{attribute 'reflection'}
FUNCTION_BLOCK Mediator
VAR_INPUT

	MoverArray				: ARRAY [1..Param.MAX_MOVERS] OF POINTER TO Mover;
	
	MoverListArray			: ARRAY [0..Param.MAX_MOVERLISTS-1] OF POINTER TO MoverList;
	PositionTriggerArray	: ARRAY [0..Param.MAX_POSITIONTRIGGERS-1] OF POINTER TO PositionTrigger;
	StationArray			: ARRAY [0..Param.MAX_STATIONS-1] OF POINTER TO Station;
	ZoneArray				: ARRAY [0..Param.MAX_ZONES-1] OF POINTER TO Zone;
	TrackArray				: ARRAY [0..Param.NUM_TRACKS] OF POINTER TO Track;	// track 0 is a special absolute case, this makes the array 1 larger than normal	

	GROUP_REF				: AXES_GROUP_REF;
	
END_VAR
VAR_OUTPUT
	Error			: BOOL;			// error is currently active
	ErrorID			: UDINT;		// errorID of the active error
	ErrorOrigin		: STRING;		// error source, in case of errored internal function block
	NumMovers		: USINT;		// number of movers in system
END_VAR
VAR
	{attribute 'instance-path'}
	{attribute 'noinit'}
	{attribute 'hide'}
	internalInstancePath		: STRING;	// instance naming, for diagnostics purposes

	internalMoverList				: MoverList;
	internalMoverListRecalc			: BOOL;
	internalM1DetectFlag			: BOOL;
	internalM1DetectState			: INT;
	internalEnableGroupFlag			: BOOL;
	internalEnableGroupState		: INT;
	internalEnabled					: BOOL;
	internalMover1Error				: BOOL;
	
	// implements memoization of Mediator.AllMotorModulesReady
	// so it is only computed once per scan when needed
	internalMotorModuleEnabled		:  MotorModuleStatus_typ;
	internalMotorModule48v			:  MotorModuleStatus_typ;

	// ========= XTS Utility Diagnostics =========
	fbXtsEnvironment				: FB_TcIoXtsEnvironment;
	fbXtsEnvironmentVisu			: FB_XtsEnvironmentVisu;
	nEnvironmentState				: INT;
	internalInfoServerOTCID			: UDINT;

	internalEnvironment				: I_TcIoXtsEnvironment;
	internalXPU						: I_TcIoXtsProcessingUnit;
	internalInfoServer				: I_TcIoXtsInfoServer;
	internalInfoServerCount			: UINT;
	
	// ========= internal function blocks =========
	fbGroupStatus			: MC_GroupReadStatus;
	fbGroupEnable			: MC_GroupEnable;
	fbGroupReset			: MC_GroupReset;
	fbGroupStop				: MC_GroupStop;

END_VAR
VAR CONSTANT
	ADD_TO_GROUP_SIZE		: UDINT := 30;
END_VAR

METHOD AddMover : BOOL
VAR_INPUT
	
	Mover		: REFERENCE TO Mover;

END_VAR

VAR
	duplicateFound		: BOOL;
	i					: DINT;
	emptyIDX			: DINT := -1;;
END_VAR


// Check for duplicates

IF __ISVALIDREF( Mover ) THEN
	
	Mover.Mediator			REF= THIS^;

	duplicateFound			:= FALSE;
	
	FOR i := 1 TO SIZEOF( MoverArray ) / SIZEOF( MoverArray[1] ) DO
		IF MoverArray[i] <> 0 THEN		// verify the element is clear to prevent overwrites
			IF ADR(Mover) = MoverArray[i] THEN
				duplicateFound		:= TRUE;	// this mover is already mediated
			END_IF
		ELSE
			// track the first empty index
			IF (emptyIDX = -1) THEN
				emptyIDX	:= i;
			END_IF;
		END_IF	
	END_FOR
	
	// if no empty index is available set a message and return
	IF emptyIDX = -1 THEN
		ADSLOGSTR( ADSLOG_MSGTYPE_WARN, 'AddMover System Array is full. %s not added. Check Params.MAX_MOVERS' , Mover.InstancePath);
		RETURN;
	END_IF;
	
	IF duplicateFound = FALSE THEN
		
		THIS^.MoverArray[emptyIDX]		:= ADR( Mover );	// new mover into empty array element

		// Automatically register the mover with any Position Triggers
		FOR i := 0 TO SIZEOF( PositionTriggerArray ) / SIZEOF( PositionTriggerArray[0] ) - 1 DO
			IF PositionTriggerArray[i] <> 0 THEN
				PositionTriggerArray[i]^.RegisterMover( Mover );
			END_IF			
		END_FOR
		
		// Automatically register the mover with any Zones
		FOR i := 0 TO SIZEOF( ZoneArray ) / SIZEOF( ZoneArray[0] ) - 1 DO
			IF ZoneArray[i] <> 0 THEN
				ZoneArray[i]^.RegisterMover( Mover );
			END_IF
		END_FOR
		
	END_IF
END_IF

// set the flag to recalculate the internal mover list
internalMoverListRecalc := TRUE;
END_METHOD

METHOD AddMoverList : BOOL
VAR_INPUT
	
	MoverList		: REFERENCE TO MoverList;

END_VAR

VAR
	duplicateFound		: BOOL;
	i					: DINT;
	emptyIDX			: DINT := -1;
END_VAR


// Check for duplicates
IF __ISVALIDREF( MoverList ) THEN
	
	MoverList.Mediator			REF= THIS^;
	
	duplicateFound				:= FALSE;
	
	FOR i := 0 TO SIZEOF( MoverListArray ) / SIZEOF( MoverListArray[0] ) - 1 DO
		IF MoverListArray[i] <> 0 THEN		// verify the element is clear to prevent overwrites
			IF ADR( MoverList ) = MoverListArray[i] THEN
				duplicateFound		:= TRUE;		// this moverlist is already mediated
			END_IF
		ELSE
			// track the first empty index
			IF (emptyIDX = -1) THEN
				emptyIDX	:= i;
			END_IF;
		END_IF
	END_FOR
	
	// if no empty index is available set a message and return
	IF emptyIDX = -1 THEN
		ADSLOGSTR( ADSLOG_MSGTYPE_WARN, 'MoverList System Array is full. %s not added. Check Params.MAX_MOVERLISTS' , MoverList.InstancePath);
		RETURN;
	END_IF;
	
	IF duplicateFound = FALSE THEN
		THIS^.MoverListArray[emptyIDX]		:= ADR( MoverList );
	END_IF
END_IF

// set the flag to recalculate the internal mover list
internalMoverListRecalc := TRUE;
END_METHOD

METHOD AddPositionTrigger : BOOL
VAR_INPUT
	
	PositionTrigger		: REFERENCE TO PositionTrigger;

END_VAR

VAR
	duplicateFound		: BOOL;
	i					: DINT;
	emptyIDX			: DINT := -1;
END_VAR


// Check for duplicates
IF __ISVALIDREF( PositionTrigger ) THEN
	
	PositionTrigger.Mediator		REF= THIS^;
	
	duplicateFound					:= FALSE;
	
	FOR i := 0 TO SIZEOF( PositionTriggerArray ) / SIZEOF( PositionTriggerArray[0] ) - 1 DO
		IF PositionTriggerArray[i] <> 0 THEN		// verify the element is clear to prevent overwrites
			IF ADR( PositionTrigger ) = PositionTriggerArray[i] THEN
				duplicateFound		:= TRUE;		// this moverlist is already mediated
			END_IF
		ELSE
			// track the first empty index
			IF (emptyIDX = -1) THEN
				emptyIDX	:= i;
			END_IF;
		END_IF
	END_FOR
	
	// if no empty index is available set a message and return
	IF emptyIDX = -1 THEN
		ADSLOGSTR( ADSLOG_MSGTYPE_WARN, 'AddPositionTrigger System Array is full. %s not added. Check Params.MAX_POSITIONTRIGGERS' , PositionTrigger.InstancePath);
		RETURN;
	END_IF;
	
	IF duplicateFound = FALSE THEN
		THIS^.PositionTriggerArray[emptyIDX]		:= ADR( PositionTrigger );
		
		// Automatically register all existing movers with the new position trigger
		FOR i := 1 TO SIZEOF( MoverArray ) / SIZEOF( MoverArray[1] ) DO
			IF MoverArray[i] <> 0 THEN
				THIS^.PositionTriggerArray[emptyIDX]^.RegisterMover( MoverArray[i]^ );
			END_IF
		END_FOR		
		
	END_IF
END_IF
END_METHOD

METHOD AddStation : BOOL
VAR_INPUT
	
	Station		: REFERENCE TO Station;

END_VAR

VAR
	duplicateFound		: BOOL;
	i					: DINT;
	emptyIDX			: DINT := -1;
END_VAR


// Check for duplicates
IF __ISVALIDREF( Station ) THEN
	
	Station.Mediator	REF= THIS^;
	
	duplicateFound		:= FALSE;
	
	FOR i := 0 TO SIZEOF( StationArray ) / SIZEOF( StationArray[0] ) - 1 DO
		IF StationArray[i] <> 0 THEN		// verify the element is clear to prevent overwrites
			IF ADR( Station ) = StationArray[i] THEN
				duplicateFound		:= TRUE;		// this moverlist is already mediated
			END_IF
		ELSE
			// track the first empty index
			IF (emptyIDX = -1) THEN
				emptyIDX	:= i;
			END_IF;
		END_IF
	END_FOR
	
	// if no empty index is available set a message and return
	IF emptyIDX = -1 THEN
		ADSLOGSTR( ADSLOG_MSGTYPE_WARN, 'AddStation System Array is full. %s not added. Check Params.MAX_STATIONS' , Station.InstancePath);
		RETURN;
	END_IF;
	
	IF duplicateFound = FALSE THEN
		THIS^.StationArray[emptyIDX]		:= ADR( Station );
		// store unique index for station
		Station.Id := emptyIDX;
	END_IF
END_IF
END_METHOD

METHOD AddTrack : BOOL
VAR_INPUT
	
	Track		: REFERENCE TO Track;

END_VAR

VAR
	duplicateFound		: BOOL;
	i					: UDINT;
	emptyIDX			: UDINT;
END_VAR


// Check for duplicates
IF __ISVALIDREF( Track ) THEN
	
	Track.Mediator		REF= THIS^;
	
	duplicateFound		:= FALSE;
	
	FOR i := 0 TO SIZEOF( TrackArray ) / SIZEOF( TrackArray[0] ) - 1 DO
		IF TrackArray[i] <> 0 THEN		// verify the element is clear to prevent overwrites
			IF ADR( Track ) = TrackArray[i] THEN
				duplicateFound		:= TRUE;		// this moverlist is already mediated
			END_IF
		ELSE
			// track the first empty index
			IF (emptyIDX = 0) THEN
				emptyIDX	:= i;
			END_IF;
		END_IF
	END_FOR
	
	IF duplicateFound = FALSE THEN
		THIS^.TrackArray[emptyIDX]		:= ADR( Track );
	END_IF
END_IF
END_METHOD

METHOD AddZone : BOOL
VAR_INPUT
	
	Zone		: REFERENCE TO Zone;

END_VAR

VAR
	duplicateFound		: BOOL;
	i					: DINT;
	emptyIDX			: DINT := -1;
END_VAR


// Check for duplicates
IF __ISVALIDREF( Zone ) THEN
	
	Zone.Mediator		REF= THIS^;
	
	duplicateFound		:= FALSE;
	
	FOR i := 0 TO SIZEOF( ZoneArray ) / SIZEOF( ZoneArray[0] ) - 1 DO
		IF ZoneArray[i] <> 0 THEN		// verify the element is clear to prevent overwrites
			IF ADR( Zone ) = ZoneArray[i] THEN
				duplicateFound		:= TRUE;		// this moverlist is already mediated
			END_IF
		ELSE
			// track the first empty index
			IF (emptyIDX = -1) THEN
				emptyIDX	:= i;
			END_IF;
		END_IF
	END_FOR
	
	// if no empty index is available set a message and return
	IF emptyIDX = -1 THEN
		ADSLOGSTR( ADSLOG_MSGTYPE_WARN, 'AddZone System Array is full. %s not added. Check Params.MAX_ZONES' , Zone.InstancePath);
		RETURN;
	END_IF;
	
	IF duplicateFound = FALSE THEN
		THIS^.ZoneArray[emptyIDX]		:= ADR( Zone );
		
		// Automatically register all existing movers with the new zone
		FOR i := 1 TO SIZEOF( MoverArray ) / SIZEOF( MoverArray[1] ) DO
			IF MoverArray[i] <> 0 THEN
				THIS^.ZoneArray[emptyIDX]^.RegisterMover( MoverArray[i]^ );
			END_IF
		END_FOR
		
	END_IF
END_IF
END_METHOD

{attribute 'monitoring' := 'call'}
PROPERTY AllMotorModules48vReady : Bool
GET
VAR
	I				: UDINT;
	nParts			: UDINT;
	b48vReady	: BOOL;
	PartTcIo		: I_TcIoXtsXpuPart;
END_VAR
// this is calculation and ADS intensive so the result is memozied once per scan

// only run the sum if the calc bit has not been set for this scan
IF (NOT internalMotorModule48v.calcComplete) THEN
	// Monitor DriveStatus to disallow motion commands before high drive has been achieved.
	IF fbXtsEnvironment.P_IsInitialized THEN
	// Get number of parts. 
		nParts:= fbXtsEnvironment.XpuTcIo(1).P_PartCount;
		IF nParts <> 0 THEN
			// Get number of modules per part and check their state
			b48vReady:= TRUE;
			FOR I := 1 TO nParts DO 
				PartTcIo := fbXtsEnvironment.XpuTcIo(1).PartTcIo(UDINT_TO_UINT(I));
				// and the previous result with the result for this part
				b48vReady := b48vReady AND PartMotorModules48vReady(PartTcIo);
			END_FOR
		END_IF
	END_IF

	// memoize the result
	internalMotorModule48v.calcResult := b48vReady;
	internalMotorModule48v.calcComplete := TRUE;
END_IF;

// return the result
AllMotorModules48vReady:= internalMotorModule48v.calcResult;
END_GET
END_PROPERTY

{attribute 'monitoring' := 'call'}
PROPERTY AllMotorModulesEnabled : Bool
GET
VAR
	I				: UDINT;
	nParts			: UDINT;
	bHighDriveReady	: BOOL;
	PartTcIo		: I_TcIoXtsXpuPart;
END_VAR
// this is calculation and ADS intensive so the result is memozied once per scan

// only run the sum if the calc bit has not been set for this scan
IF (NOT internalMotorModuleEnabled.calcComplete) THEN
	// Monitor DriveStatus to disallow motion commands before high drive has been achieved.
	IF fbXtsEnvironment.P_IsInitialized THEN
	// Get number of parts. 
		nParts:= fbXtsEnvironment.XpuTcIo(1).P_PartCount;
		IF nParts <> 0 THEN
			// Get number of modules per part and check their state
			bHighDriveReady:= TRUE;
			FOR I := 1 TO nParts DO 
				PartTcIo := fbXtsEnvironment.XpuTcIo(1).PartTcIo(UDINT_TO_UINT(I));
				// and the previous result with the result for this part
				bHighDriveReady := bHighDriveReady AND PartMotorModulesEnabled(PartTcIo);
			END_FOR
		END_IF
	END_IF

	// memoize the result
	internalMotorModuleEnabled.calcResult := bHighDriveReady;
	internalMotorModuleEnabled.calcComplete := TRUE;
END_IF;

// return the result
AllMotorModulesEnabled:= internalMotorModuleEnabled.calcResult;
END_GET
END_PROPERTY

PROPERTY CompleteMoverList : iMoverList
GET
VAR
	i: UDINT;
END_VAR
// the mover list is populated in cyclic when needed
// flags in the methods .AddMover and .AddMoverList trigger the recalculation

CompleteMoverList	:= internalMoverList;
END_GET
END_PROPERTY

METHOD Cyclic : BOOL
VAR_INPUT
	NUM_MOVERS			: USINT;
END_VAR

VAR
	eMoverIdDetectionMode : MoverIdDetectionMode;
	eMoverIdDetectionState : MoverIdDetectionStateEnum;
END_VAR

VAR_INST
	MsgCreate		: FB_TcMessage;
	
	// station info state machine support
	nInfoServerState : INT;
	PartStartEnd : ARRAY [1..Param.PART_ARRAY_SIZE] OF ARRAY [0..1] OF LREAL;
	nPartsInTrack1	: UDINT;
	TrackPartInfo	: ARRAY[1..TcIoXtsEnvironmentParameterList.MaxPartsPerTrack] OF ST_PartInfoItems;
	PartInfo 		: St_PartInfoItems;
	nInfoServerStations		: UDINT;
	nUsableStations			: UDINT;
	StationTcIo		: I_TcIoXtsInfoServerInfoStation;
	nStationPartNum	: UDINT;
	pXtsStation		: POINTER TO Station;
	PartObjectIds	: ARRAY [1..TcIoXtsEnvironmentParameterList.MaxXtsPartsPerXpu] OF OTCID;
	StopPositions	: ARRAY [1..TcIoXtsEnvironmentParameterList.MaxXtsStopPositionsPerStation] OF LREAL := [0.0];
	i				: UDINT;
	j				: UDINT;
	workingStation	: UDINT;
	
	XPUDetectionState	: DetectionStateEnum;
END_VAR
// this method contains multiple state machines denoted by the headers below

// update output data
NumMovers := NUM_MOVERS;

// clear memoized values for recalculation
internalMotorModuleEnabled.calcComplete := FALSE;
internalMotorModule48v.calcComplete := FALSE;

// regenerate the internal mover list when necessary
IF (internalMoverListRecalc) THEN
	// this is returned by the property CompleteMoverList, and does not need to be calculated on every call to the property
	// reset flag
	internalMoverListRecalc := FALSE;
	// clear the list
	internalMoverList.UnregisterAll();
	// re-populate the list
	FOR i := 1 TO SIZEOF( MoverArray ) / SIZEOF( MoverArray[1] ) DO
		IF MoverArray[i] <> 0 THEN
			internalMoverList.RegisterMover( MoverArray[i]^ );
		END_IF
	END_FOR
END_IF

// Handle all project cyclic calls

FOR i := 1 TO Param.MAX_MOVERS DO
	IF MoverArray[i] <> 0 THEN
		// handle cyclic calls
		MoverArray[i]^.Cyclic( GROUP_REF );			// could make this ca group addition clener
		MoverArray[i]^.AxisReference.ReadStatus();
		MoverArray[i]^.MoverIndex := i;
	END_IF
END_FOR

FOR i := 0 TO Param.MAX_STATIONS - 1 DO
	IF StationArray[i] <> 0 THEN
		StationArray[i]^.Cyclic();
	END_IF
END_FOR

FOR i := 0 TO Param.MAX_POSITIONTRIGGERS - 1 DO
	IF PositionTriggerArray[i] <> 0 THEN
		PositionTriggerArray[i]^.Cyclic();
	END_IF
END_FOR

FOR i := 0 TO Param.NUM_TRACKS DO
	IF TrackArray[i] <> 0 THEN
		TrackArray[i]^.Cyclic();
	END_IF
END_FOR

// *************************************************************************
// environment state machine
// *************************************************************************

CASE nEnvironmentState OF
	0:	// ----------------------------------------- Enable Init Items
	
		// the procedure for initializing the XTS environment has changed
		// this step previously held configuration values for the environment
		// it is left as a placeholder for consistency with additional steps below
		
		// Next step
		nEnvironmentState	:= 1;
		
	1:	// ------------------------------------------ Init Environment
		
		// Start init
		IF fbXtsEnvironment.Init(TRUE) THEN
			// stop init
			fbXtsEnvironment.Init(FALSE);
			
			// next step
			nEnvironmentState	:= 2;
		END_IF
		
	2:	// ------------------------------------------ Check for success
	
		// Check IsInitialized property
		IF fbXtsEnvironment.P_IsInitialized THEN
			// assign to vars
			internalEnvironment 	:= fbXtsEnvironment;
			internalXPU				:= fbXtsEnvironment.XpuTcIo(1);
			internalInfoServerCount := fbXtsEnvironment.P_InfoServerCount;
			// info server may not be present in hand-built XTS configurations
			IF (internalInfoServerCount > 0) THEN
				internalInfoServer	:= fbXtsEnvironment.InfoServerTcIo(1);
				nEnvironmentState := 3;
			ELSE
				// skip info server intializiation
				nEnvironmentState := 6;
			END_IF;
		END_IF

	3:	// ------------------------------------------ Get OTCID
	
		IF internalEnvironment.GetInfoServerOids(TRUE) THEN
			internalEnvironment.GetInfoServerOids(FALSE);
			internalInfoServerOTCID := internalEnvironment.P_InfoServerOids[1];
			nEnvironmentState := 4;
		END_IF;
		
	4:	// ------------------------------------------- Init info server
		
		// Start init
		IF internalInfoServer.Init(TRUE, internalInfoServerOTCID) THEN
			// stop init
			internalInfoServer.Init(FALSE, internalInfoServerOTCID);
			
			// next step
			nEnvironmentState	:= 5;
		END_IF
	5:	// ------------------------------------------ Check for success
	
		// Check IsInitialized property
		IF internalInfoServer.P_IsInitialized THEN
			// next step
			nEnvironmentState	:= 6;
		END_IF
		
	6:	// ------------------------------------------- Init Visu
	
		fbXtsEnvironmentVisu( ipTcIoXtsEnvironment := fbXtsEnvironment );
		
		// next step
		nEnvironmentState	:= 7;
		
	7:	// ------------------------------------------- Init done

		fbXtsEnvironmentVisu.Cycle();
		
END_CASE

// *************************************************************************
// mover 1 detection state machine
// *************************************************************************

// monitor for the group reset flag and act on it
CASE internalM1DetectState OF 
	0:	// wait for flag
		IF internalM1DetectFlag THEN
			// clear previous error flag
			internalMover1Error		:= FALSE;
			internalM1DetectState	:= 10;
		END_IF
		
	10:	// wait for envrionment
		IF EnvironmentIsReady AND_THEN NOT THIS^.Mover1DetectionComplete THEN
 			internalM1DetectState 	:= 20;
		END_IF

	20:	// Trigger mover redetection
		fbXtsEnvironment.XpuTcIo(1).TriggerRedetection();
 		internalM1DetectState 		:= 30;

	30:	// Monitor mover redection status
		XPUDetectionState			:= fbXtsEnvironment.XpuTcIo(1).GetDetectionState();
		IF XPUDetectionState = DetectionStateEnum.Succeeded THEN
			internalM1DetectState 	:= 40;
		ELSIF XPUDetectionState > DetectionStateEnum.Succeeded THEN
			internalM1DetectState	:= 900;
		END_IF

		(*	DetectionStateEnum: NotStarted:=0, 
								Running:=1,
								Succeeded:=2,
								FailedDueToEnabledMovers:=3,
								FailedExpectedMoversNotDetected:=4,
								FailedNotEnoughMovers:=5,
								FailedNoTracksIncluded:=6,
								FailedTooManyActiveMovers:=7) 	*)

	40:	// check for mover 1 mode
		eMoverIdDetectionMode := XPU.GetMoverIdDetectionMode();
		IF (eMoverIdDetectionMode = MoverIdDetectionMode.Mover1 OR eMoverIdDetectionMode = MoverIdDetectionMode.MultipleMover1) THEN
			// mover 1 detection sequence
			internalM1DetectState := 100;
		ELSE
			// no detection required
			internalM1DetectState := 200;
		END_IF
		
	100: // check if mover 1 id is avtive
		eMoverIdDetectionState := XPU.GetMoverIdDetectionState();
		IF (eMoverIdDetectionState <> MoverIdDetectionStateEnum.Valid) THEN
			// start the detection
			XPU.TriggerMoverIdDetection();
		END_IF;
		internalM1DetectState := 110;
		
	110: // wait for group detection results
		eMoverIdDetectionState := XPU.GetMoverIdDetectionState();
		IF eMoverIdDetectionState = MoverIdDetectionStateEnum.Error THEN
			// error state
			internalM1DetectState := 900;
		ELSIF eMoverIdDetectionState = MoverIdDetectionStateEnum.Valid THEN
			// detection complete
			internalM1DetectState := 200;
		END_IF;
				
	
	200: // set flags and clean up
		// flag is read directly from XPU in Mover1DetectionComplete property
		internalM1DetectState := 0;
	
	900:
		// error state
		// set error flag for movers to respond
		internalMover1Error := TRUE;
		// send message
		MsgCreate.CreateEx( TC_EVENTS.XtsBaseEventClass.Mover1Detection,0 );
		MsgCreate.ipArguments.Clear();
		MsgCreate.Send(0);
		// return to idle
		internalM1DetectState := 0;
		
		
END_CASE

// reset flag always
internalM1DetectFlag := FALSE;

// *************************************************************************
// group enable state machine
// *************************************************************************

// get group status for property
fbGroupStatus.Enable := TRUE;
fbGroupStatus( AxesGroup := GROUP_REF );

CASE internalEnableGroupState OF
	0:	// wait for flag 
		IF internalEnableGroupFlag AND NOT internalEnabled THEN
			internalEnableGroupState := 10;
			Error := FALSE;
		END_IF;

	10: // ------------------------------------------------------- check the status of the group
	
		IF fbGroupStatus.Valid AND fbGroupStatus.GroupErrorStop THEN
			fbGroupReset.Execute		:= TRUE;
		ELSIF fbGroupStatus.Valid AND fbGroupStatus.GroupDisabled THEN
			fbGroupReset.Execute		:= FALSE;
			internalEnableGroupState	:= 20;
		ELSIF fbGroupStatus.Valid AND ( fbGroupStatus.GroupStandby OR fbGroupStatus.GroupMoving ) THEN
			fbGroupReset.Execute		:= FALSE;
			internalEnableGroupState	:= 100;
		END_IF
		
		IF fbGroupStatus.Error THEN
			fbGroupReset.Execute		:= FALSE;
			ErrorID						:= fbGroupStatus.ErrorId;
			ErrorOrigin					:= CONCAT( internalInstancePath, '.fbGroupStatus' );
			MsgCreate.CreateEx( TC_EVENTS.XtsBaseEventClass.fbGroupStatus,0 );
			MsgCreate.ipArguments.Clear().AddString(THIS^.internalInstancePath).AddUDINT(THIS^.ErrorID);
			internalEnableGroupState	:= 900;
		ELSIF fbGroupReset.Error THEN
			fbGroupReset.Execute		:= FALSE;
			ErrorID						:= fbGroupReset.ErrorId;
			ErrorOrigin					:= CONCAT( internalInstancePath, '.fbGroupReset' );
			MsgCreate.CreateEx( TC_EVENTS.XtsBaseEventClass.fbGroupReset,0 );
			MsgCreate.ipArguments.Clear().AddString(THIS^.internalInstancePath).AddUDINT(THIS^.ErrorID);
			internalEnableGroupState	:= 900;
		END_IF
		
	
	20: // ------------------------------------------------------- enable the group
		
		fbGroupEnable.Execute			:= TRUE;
		
		IF fbGroupEnable.Done AND GROUP_REF.NcToPlc.CA.Common.GroupStatus.State = mcGroupStateStandby AND fbGroupStatus.GroupErrorStop = FALSE THEN
			fbGroupEnable.Execute		:= FALSE;
			internalEnableGroupFlag 	:= FALSE;
			internalEnableGroupState	:= 100;
		ELSIF fbGroupEnable.Error THEN
			fbGroupEnable.Execute		:= FALSE;
			ErrorID						:= fbGroupEnable.ErrorId;
			ErrorOrigin					:= CONCAT( internalInstancePath, '.fbGroupEnable' );
			MsgCreate.CreateEx( TC_EVENTS.XtsBaseEventClass.fbGroupEnable,0 );
			MsgCreate.ipArguments.Clear().AddString(THIS^.internalInstancePath).AddUDINT(THIS^.ErrorID);
			MsgCreate.Send(0);
			internalEnableGroupState	:= 900;
		END_IF
		
	100: // clean up flags and rewind
		internalEnabled 				:= TRUE;
		internalEnableGroupState 		:= 0;
		
	900: // error
		Error 							:= TRUE;
		internalEnabled 				:= FALSE;
		IF NOT internalEnableGroupFlag THEN
			Error						:= FALSE;
			ErrorID						:= 0;
			ErrorOrigin					:= '';
			internalEnableGroupState	:= 0;
		END_IF
		
END_CASE

internalEnableGroupFlag := FALSE;

// catch error flag and reset custom status bit
IF (fbGroupStatus.GroupErrorStop AND internalEnableGroupState = 0 AND internalEnabled) THEN
	Error := TRUE;
	internalEnabled := FALSE;
END_IF

// cyclic calls
fbGroupEnable( AxesGroup := GROUP_REF );
fbGroupReset( AxesGroup := GROUP_REF );
fbGroupStop( AxesGroup := GROUP_REF );

// always clear the triggering flag
//internalEnableGroupFlag := FALSE;

// *************************************************************************
// station info state machine
// *************************************************************************

// populate TcCom XTS station objects with positions and part numbers from code for easier visibility in simulation

// check for environment
IF THIS^.InfoServerIsReady AND internalEnabled AND Param.AUTO_POPULATE_STATIONS THEN
	
	CASE nInfoServerState OF
		
	// get number of parts via track 1 and store start/end positions in 
		0:
			// check for defined track in first position
			IF (internalXPU.P_TrackCount >= 1) THEN
				nInfoServerState := 10;
			END_IF
			
		10:
			// get info about array of parts
			nPartsInTrack1 := internalXPU.TrackTcIo(1).GetPartCount();
			nInfoServerState := 20;
			
		20:
			// get info for each part start and end position (or max size of array)
			TrackPartInfo := internalXPU.TrackTcIo(1).GetPartInfoItems();
			FOR i := 1 TO MIN(nPartsInTrack1, Param.PART_ARRAY_SIZE) DO
				PartInfo := TrackPartInfo[i];
				PartStartEnd[i][0] := PartInfo.fOffset;
				PartStartEnd[i][1] := PartInfo.fLength + PartInfo.fOffset;
			END_FOR
			nInfoServerState := 30;

		30:
			// get number of stations
			nInfoServerStations := internalInfoServer.GetInfoStationCount() ;
			nInfoServerStations := internalINfoServer.P_InfoStationCount;
			nInfoServerState := 40;
			
		40:
			// calculate minimum number of stations that can be set up
			nUsableStations := MIN(nInfoServerStations, Param.MAX_STATIONS);
			workingStation := 0;
			FOR i := 1 TO nUsableStations DO
				workingStation := workingStation + 1;
				// in case a sparse Station array is used, only detect stations that have a position value <> 0
				WHILE (workingStation < Param.MAX_STATIONS AND_THEN (StationArray[workingStation] = 0 OR_ELSE StationArray[workingStation]^.Position = 0)) DO
					workingStation := workingStation + 1;
				END_WHILE
				// check for valid working station, and exit this for loop iteration if we're outside it
				IF workingStation >= Param.MAX_STATIONS THEN
					EXIT;
				END_IF
				// get XTS_Base Station pointer
				pXtsStation := StationArray[workingStation];
				// test for valid pointer (station has been through the Mediator.AddStation method)
				IF (pXtsStation <> 0) THEN
					// make sure the position is not zero (hides stations that probably aren't used)
						IF (pXtsStation^.Position <> 0.0) THEN
						// calculate part number
						nStationPartNum := 0;
						FOR j := 1 TO nPartsInTrack1 DO
							IF (PartStartEnd[j][0] <= pXtsStation^.Position AND pXtsStation^.Position < PartStartEnd[j][1]) THEN
								nStationPartNum := j;
							END_IF
						END_FOR
						// test for found part number
						IF (nStationPartNum > 0) THEN
						// get station
							StationTcIO := internalInfoServer.InfoStationTcIo(UDINT_TO_UINT(i));
							// test for valid station
							IF (stationTcIO <> 0) THEN
								// write station tc io object back to XTS.Station for later use
								pXtsStation^.StationTcIo := StationTcIO;
								// try not to overwrite data that may have been entered in the configurator by testing for a start position of 0 (from the configurator), or 10 and 200 (defaults from adding object by hand)
								IF (StationTcIO.GetStartPositionOnPart() = 0.0 OR (StationTcIO.GetStartPositionOnPart() = 10.0 AND StationTcIO.GetEndPositionOnPart() = 200.0)) THEN
									// assign data
									StationTcIO.SetStationId(i);
									PartObjectIds[1] := TrackPartInfo[nStationPartNum].nObjectId;
									stationTcIO.SetPartObjectIds(PartObjectIds);
									StationTcIO.SetStartPositionOnPart(pXtsStation^.Position - PartStartEnd[nStationPartNum][0]);
									StationTcIO.SetEndPositionOnPart(pXtsStation^.Position - PartStartEnd[nStationPartNum][0]);
									StationTcIo.SetStopPositions(StopPositions);
									StationTcIo.SetStationColor(16#FFEF0000);	// Beckhoff red
									StationTcIO.SetIsEnabled(TRUE);	// v4.x "dims" the color of disabled stations
									StationTcIO.SetDescription(pXtsStation^.Description);
								END_IF;
							END_IF;
						END_IF;
					END_IF;
				END_IF;
			END_FOR
			// transition to non-existent state. This routine only runs one time at the first enable signal.
			nInfoServerState := 50;
	END_CASE
END_IF
END_METHOD

METHOD DetectMover1 : BOOL
VAR_INPUT
END_VAR
// calling enable group only sets a group reset flag that is handled in Cyclic Group Reset
// this effectively sums up requests from all movers into a single sequence that will handle the reset
internalM1DetectFlag := TRUE;
END_METHOD

METHOD DisableGroup : BOOL
VAR_INPUT
END_VAR
// reset the internal group enable flag so the enable sequence in mediator.cyclic is re-armed
internalEnabled := FALSE;
Error := FALSE;
END_METHOD

METHOD EnableGroup : BOOL
VAR_INPUT
END_VAR
// calling enable group only sets a group reset flag that is handled in Cyclic Group Reset
// this effectively sums up requests from all movers into a single sequence that will handle the reset
internalEnableGroupFlag := TRUE;
END_METHOD

PROPERTY Environment : I_TcIoXtsEnvironment
GET
Environment := internalEnvironment;
END_GET
END_PROPERTY

{attribute 'monitoring' := 'call'}
PROPERTY EnvironmentIsReady : BOOL
GET
// was fbXtsEnvironment.P_IsInitialized, but this can error if fbXtsEnironment.Init has not yet returned true
// the state of the environment state machine is now used to confirm init has ben called
EnvironmentIsReady := nEnvironmentState >= 3;
END_GET
END_PROPERTY

{attribute 'monitoring' := 'call'}
PROPERTY GroupAddLimit : UDINT
GET
// when adding movers to gropus, a smaller subset of movers should be added, not all at once
// this returns the highest mover number that can currently be added to the group
// based on the size of the add_to_group constant

// with a size limit of 30 this will return 30, then 60, 90 etc (30 at a time, with 1-based mover array)
// deliberate integer math is used to truncate the quotent of the group step check
GroupAddLimit := (REAL_TO_UDINT(UDINT_TO_REAL(GROUP_REF.NcToPlc.CA.Common.GroupAxesCount)/UDINT_TO_REAL(ADD_TO_GROUP_SIZE))+1)*ADD_TO_GROUP_SIZE;
END_GET
END_PROPERTY

{attribute 'monitoring' := 'call'}
PROPERTY GroupAxesCount : UDINT
GET
GroupAxesCount := GROUP_REF.NcToPlc.CA.Common.GroupAxesCount;
END_GET
END_PROPERTY

{attribute 'monitoring' := 'call'}
PROPERTY GroupEnabled : bool
GET
{attribute 'monitoring' := 'call'}
VAR
END_VAR
GroupEnabled := internalEnabled;
END_GET
END_PROPERTY

{attribute 'monitoring' := 'call'}
PROPERTY GroupError : bool
GET
{attribute 'monitoring' := 'call'}
VAR
END_VAR
// sum of various error bits throughout the mediator
GroupError := fbGroupStatus.GroupErrorStop;
END_GET
END_PROPERTY

PROPERTY InfoServer : I_TcIoXtsInfoServer
GET
InfoServer := internalInfoServer;
END_GET
END_PROPERTY

{attribute 'monitoring' := 'call'}
PROPERTY InfoServerIsReady : BOOL
GET
InfoServerIsReady := internalInfoServer <> 0 AND_THEN internalInfoServer.P_IsInitialized;
END_GET
END_PROPERTY

{attribute 'monitoring' := 'call'}
PROPERTY InstancePath : string
GET
InstancePath := internalInstancePath;
END_GET
END_PROPERTY

{attribute 'monitoring' := 'call'}
PROPERTY Mover1DetectionComplete : BOOL
GET
{attribute 'monitoring' := 'call'}
VAR
END_VAR
Mover1DetectionComplete := THIS^.EnvironmentIsReady AND_THEN XPU.GetMoverIdDetectionState() = MoverIdDetectionStateEnum.Valid;
END_GET
END_PROPERTY

{attribute 'monitoring' := 'call'}
PROPERTY Mover1DetectionError : bool
GET
{attribute 'monitoring' := 'call'}
VAR
END_VAR
Mover1DetectionError := internalMover1Error;
END_GET
END_PROPERTY

METHOD MuteAllPositionTriggers : BOOL
VAR_INPUT
END_VAR
VAR
	i : UDINT;
END_VAR
FOR i := 0 TO Param.MAX_POSITIONTRIGGERS-1 DO
	IF PositionTriggerArray[i] <> 0 THEN
		PositionTriggerArray[i]^.MuteCurrent();
	END_IF
END_FOR
END_METHOD

METHOD PartMotorModules48vReady : BOOL
VAR_INPUT
	PartTcIo		: I_TcIoXtsXpuPart;
END_VAR
VAR
END_VAR
// protect against no part provided
IF (PartTcIo = 0) THEN
	// this part can't be ready
	PartMotorModules48vReady := FALSE;
	RETURN;
END_IF

PartMotorModules48vReady := PartTcIo.GetIsDcLinkVoltageReady();
END_METHOD

METHOD PartMotorModulesEnabled : BOOL
VAR_INPUT
	PartTcIo		: I_TcIoXtsXpuPart;
END_VAR
VAR
END_VAR
// protect against no part provided
IF (PartTcIo = 0) THEN
	// this part can't be ready
	PartMotorModulesEnabled := FALSE;
	RETURN;
END_IF

PartMotorModulesEnabled := PartTcIO.GetAreAllModulesInOp();
END_METHOD

METHOD ResetStatistics : BOOL
VAR
	i					: UDINT;
END_VAR
// reset statistics at all postion triggers and stations
FOR i := 0 TO Param.MAX_POSITIONTRIGGERS-1 DO
	IF PositionTriggerArray[i] <> 0 THEN
		PositionTriggerArray[i]^.ResetStatistics();
	END_IF
END_FOR
FOR i := 0 TO Param.MAX_STATIONS-1 DO
	IF StationArray[i] <> 0 THEN
		StationArray[i]^.ResetStatistics();
	END_IF
END_FOR
END_METHOD

PROPERTY XPU : I_TcIoXtsProcessingUnit
GET
XPU := internalXPU;
END_GET
END_PROPERTY

END_FUNCTION_BLOCK

(* stored: Version 1.1.0.1, ProductVersion 3.1.4026.18
   POU Mediator: Id {164d51b4-07ec-0e46-0eb0-392af39d7d3a}, SpecialFunc None
   Folder Methods: Id {0d177045-c92a-0627-14e7-41e4c9da72c3}
   Folder Properties: Id {d9d81742-b9bd-0437-3780-4a446062d311}
   Method AddMover: Id {3437c27c-dd7b-0ac3-07a2-d432fc68235a}
   Method AddMoverList: Id {fa372345-a99c-01d2-2d94-cc2fd6bab53d}
   Method AddPositionTrigger: Id {37697d0e-c381-0846-3d01-3d7f2d276ad1}
   Method AddStation: Id {158bfd8c-35c0-05f6-1398-0d0a087d099a}
   Method AddTrack: Id {1f5fda23-0b4f-059d-05b7-42b4aba73321}
   Method AddZone: Id {b7275e17-ff08-069c-32b8-5e7a13dacb64}
   Property AllMotorModules48vReady: Id {2499191c-7efc-00ea-283b-811d27cdd608}
   Get Get: Id {f41a50ed-5c36-04fd-1f3c-454c5cf177f1}
   Property AllMotorModulesEnabled: Id {e4a76f20-75da-0820-2f6d-be0ad375c645}
   Get Get: Id {f8eb48d2-a530-04d2-2b29-7da0e49d088b}
   Property CompleteMoverList: Id {41f8f92e-6d81-02a1-048b-3da9baf27ff9}
   Get Get: Id {0ba48769-41e2-05d1-1ed6-465e4a354ad7}
   Method Cyclic: Id {f2264867-ad86-0c96-3c42-ade0fe3bf9e2}
   Method DetectMover1: Id {1d387785-e892-0967-22d4-73d2923e67ae}
   Method DisableGroup: Id {2c20cfe4-2326-0db3-0e15-8e6727fd803f}
   Method EnableGroup: Id {a75c02a5-1ca0-0df7-3f91-6bd402a249c4}
   Property Environment: Id {5e5f4ba6-ff8f-0396-2883-6b9b059dc7fd}
   Get Get: Id {67009401-6b19-0292-3a1b-93904af08df3}
   Property EnvironmentIsReady: Id {45272fae-93d1-0503-0b16-fd82b7738745}
   Get Get: Id {c1e17dfb-61a0-0ba8-0903-93fde5311796}
   Property GroupAddLimit: Id {65a16f3c-a017-0638-2d93-2d84b50013fb}
   Get Get: Id {7d2e7f70-ceaa-0c78-163f-9558b7d4e0a1}
   Property GroupAxesCount: Id {dec55c77-f258-0789-1555-26b4067cbe34}
   Get Get: Id {543f3341-ee3d-0bd4-30a4-c2f38c04ed3d}
   Property GroupEnabled: Id {dca70979-fee3-0f39-3528-000ca64a8f22}
   Get Get: Id {a4a17b6e-a2a8-0398-0745-96cf710d270e}
   Property GroupError: Id {3ac97d16-5fe4-0a9a-3305-6d88385b660b}
   Get Get: Id {faa6b223-287a-0e59-1c37-f312dffb5ec6}
   Property InfoServer: Id {816a507a-b5f1-077f-3d31-6cc9a0af8cb5}
   Get Get: Id {880f5fd5-5a90-005a-341d-63c8b7f4f011}
   Property InfoServerIsReady: Id {4e305043-af78-0914-0db5-c677c55227ed}
   Get Get: Id {8b9f3051-e0e9-0ebe-0aa7-9041fdaa0bf8}
   Property InstancePath: Id {bb75667d-d680-0397-38c7-96136879329d}
   Get Get: Id {b9a804e4-bca0-0f1c-39b3-bb2c5353dcf1}
   Property Mover1DetectionComplete: Id {b3d53d33-3d35-07f8-35ed-d0dbe454a97c}
   Get Get: Id {e92705b4-cdc3-0cc7-25dc-0275953572ce}
   Property Mover1DetectionError: Id {75004eac-41b5-0213-3156-b53daed26144}
   Get Get: Id {e224f7d4-69bc-07c0-2d34-8a91c1a73da1}
   Method MuteAllPositionTriggers: Id {bc0b53da-8e8f-05bf-3533-9a0a07403ca4}
   Method PartMotorModules48vReady: Id {98a45699-b0a3-05f3-058d-be5a14452817}
   Method PartMotorModulesEnabled: Id {b8e95bc3-b41f-0254-06ff-2216e86cf91e}
   Method ResetStatistics: Id {03455d1c-c490-0e78-3526-b69b05e0917b}
   Property XPU: Id {b9694a68-ee0f-0a17-2999-0aade43c6ce4}
   Get Get: Id {fb7fa487-baed-05fa-2f8e-e167e0e16d6f} *)
